Fanuc KAREL source: kt00959.KL

PROGRAM KT00959
%NOLOCKGROUP
VAR
ENTRY:INTEGER;PNAME : STRING[80];VNAME : STRING[80];STATUS:INTEGER;VALUE : STRING[80]
BEGIN
--
--
--
--
ENTRY=0
PNAME=''
VNAME='VALUE'
SET_VAR(ENTRY,PNAME,VNAME,VALUE,STATUS)
END KT00959
